// Mitsubishi GX Works2 project: 0715WOR   PLC: Q02/Q02H

PROGRAM MAIN
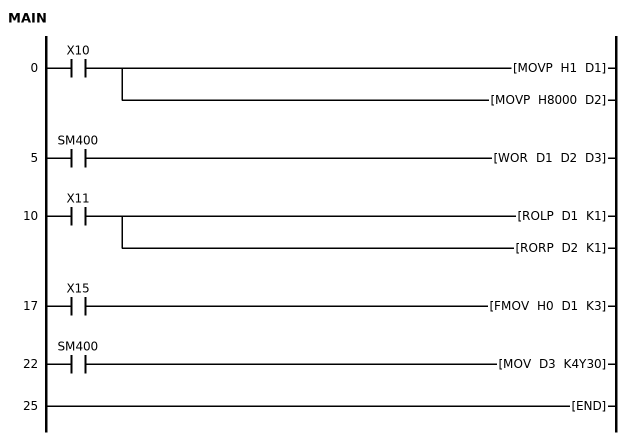
0     LD      X10
      MOVP    H1 D1
      MOVP    H8000 D2
5     LD      SM400
      WOR     D1 D2 D3
10    LD      X11
      ROLP    D1 K1
      RORP    D2 K1
17    LD      X15
      FMOV    H0 D1 K3
22    LD      SM400
      MOV     D3 K4Y30
25    END
END_PROGRAM
